// TIA Portal V18 export
// export: Created 2026-06-11T03:43:49.8808703Z, ExportSetting WithDefaults, DisplayName Totally Integrated Automation Portal, DisplayVersion V18, DisplayName TIA Portal Openness, DisplayVersion V18, DisplayName TIA Portal Version Control Interface, DisplayVersion V18, DisplayName STEP 7 Professional, DisplayVersion V18, DisplayName STEP 7 Safety, DisplayVersion V18, DisplayName WinCC Professional, DisplayVersion V18
Screen "03_PID_Muc_Nuoc"  800x600, Number=3
  ScreenLayer 
    GraphicView "Graphic view_1" at 0,0 size 800x600  Picture=Màn PID và nước
    Button "Button_1" at 27,529 size 107x46  Mode=Text, TextOff="TỔNG QUAN", TextOn="Text"
      on Click: ActivateScreen(Screen name := 01_Tong_Quan, Object number := 0)
    Button "Button_2" at 153,529 size 107x46  Mode=Text, TextOff="VẬN HÀNH", TextOn="Text"
      on Click: ActivateScreen(Screen name := 02_Van_Hanh, Object number := 0)
    Button "Button_4" at 409,528 size 107x46  Mode=Text, TextOff="TREND", TextOn="Text"
      on Click: ActivateScreen(Screen name := 04_Trend, Object number := 0)
    Button "Button_5" at 537,528 size 107x46  Mode=Text, TextOff="CẢNH BÁO", TextOn="Text"
      on Click: ActivateScreen(Screen name := 05_Canh_Bao_IO, Object number := 0)
    TextField "Text field_1" at 223,5 size 340x31  Text="MÀN HÌNH 3 - PID MỨC NƯỚC"
    Circle "Circle_3" at 677,3 size 39x39
      RangeAppearanceAnimation "RangeAppearanceAnimation"
        tag bSystemRun
        0..0: back #d9d9d9, fore #181c31
        1..1: back #00ff00, fore #181c31
    Circle "Circle_2" at 718,3 size 39x39
      RangeAppearanceAnimation "RangeAppearanceAnimation"
        tag Loi_He_Thong
        0..0: back #d9d9d9, fore #181c31
        1..1: back #ff0000, fore #181c31
    Circle "Circle_1" at 759,3 size 39x39
      RangeAppearanceAnimation "RangeAppearanceAnimation"
        tag bCheDoMoPhong
        0..0: back #d9d9d9, fore #181c31
        1..1: back #0000ff, fore #181c31
    TextField "Text field_3" at 717,42 size 43x22  Text="Fault"
    TextField "Text field_2" at 679,42 size 34x22  Text="Run"
    TextField "Text field_4" at 760,42 size 33x22  Text="Sim"
    Bar "Bar_1" at 99,165 size 93x220  CountSubDivisions=1, IntegerDigits=2, LargeTickLabelingStep=1, MaximumValue=0.5, Precision=1
      ProcessValue := Muc_Nuoc_PV
    TextField "Text field_6" at 374,80 size 30x22  Text="SP:"
    IOField "I/O field_1" at 407,82 size 37x18  DataFormat=Decimal, FormatPattern=9.9, Mode=InOutput
      ProcessValue := Muc_Nuoc_SP
    TextField "Text field_20" at 445,79 size 18x22  Text="m"
    TextField "Text field_5" at 373,112 size 30x22  Text="PV:"
    IOField "I/O field_2" at 406,114 size 40x19  DataFormat=Decimal, FormatPattern=9.9, Mode=InOutput
      ProcessValue := Muc_Nuoc_PV
    TextField "Text field_7" at 445,111 size 18x22  Text="m"
    TextField "Text field_8" at 373,144 size 32x22  Text="OP:"
    IOField "I/O field_3" at 401,144 size 49x24  DataFormat=Decimal, FormatPattern=99.9, Mode=Output
      ProcessValue := Van_Xa_OP
    TextField "Text field_9" at 443,145 size 23x22  Text="%"
    TextField "Text field_10" at 373,177 size 29x22  Text="Kp:"
    TextField "Text field_11" at 373,209 size 24x22  Text="Ti:"
    TextField "Text field_12" at 373,241 size 28x22  Text="Td:"
    IOField "I/O field_4" at 407,179 size 49x19  DataFormat=Decimal, FormatPattern=999.9, Mode=InOutput
      ProcessValue := PID_Compact_1_sRet_r_Ctrl_Gain
    IOField "I/O field_5" at 396,211 size 61x19  DataFormat=Decimal, FormatPattern=9999.9, Mode=InOutput
      ProcessValue := PID_Compact_1_sRet_r_Ctrl_Ti
    TextField "Text field_13" at 453,209 size 13x22  Text="s"
    IOField "I/O field_6" at 406,243 size 40x19  DataFormat=Decimal, FormatPattern=9.9, Mode=Output
      ProcessValue := PID_Compact_1_sRet_r_Ctrl_Td
    TextField "Text field_14" at 447,239 size 13x22  Text="s"
    Circle "Circle_4" at 486,198 size 25x25
      RangeAppearanceAnimation "RangeAppearanceAnimation"
        tag PID_Level_Enable
        0..0: back #d9d9d9, fore #181c31
        1..1: back #00ff00, fore #000000
    Circle "Circle_5" at 522,199 size 25x25
      RangeAppearanceAnimation "RangeAppearanceAnimation"
        tag Bom_Lam_Mat_M
        0..0: back #d9d9d9, fore #181c31
        1..1: back #00ccff, fore #181c31
    Circle "Circle_6" at 559,199 size 24x24
      RangeAppearanceAnimation "RangeAppearanceAnimation"
        tag Nut_EStop_HMI
        0..0: back #d9d9d9, fore #181c31
        1..1: back #00ff00, fore #181c31
    Button "Button_6" at 489,77 size 93x37  Mode=Text, TextOff="AUTO", TextOn="Text"
      RangeAppearanceAnimation "RangeAppearanceAnimation"
        tag PID_Level_Enable
        0..0: back #636571, fore #ffffff
        1..1: back #00ff00, fore #000000
      on Click: SetBit(Tag := PID_Level_Enable)
    Button "Button_7" at 489,147 size 93x37  Mode=Text, TextOff="MANUAL", TextOn="Text"
      RangeAppearanceAnimation "RangeAppearanceAnimation"
        tag PID_Level_Enable
        0..0: back #ffff00, fore #000000
        1..1: back #969696, fore #ffffff
      on Click: ResetBit(Tag := PID_Level_Enable)
    Rectangle "Rectangle_1" at 484,225 size 32x40
    TextField "Text field_15" at 481,231 size 36x24  Text="PID ENABLE"
    Rectangle "Rectangle_2" at 518,225 size 32x40
    Rectangle "Rectangle_3" at 553,225 size 32x40
    TextField "Text field_16" at 520,231 size 28x24  Text="PUMP OK"
    TextField "Text field_17" at 553,232 size 31x24  Text="ESTOP OK"
    Circle "Circle_7" at 752,169 size 13x13
      RangeAppearanceAnimation "RangeAppearanceAnimation"
        tag PID_Level_Enable
        0..0: back #d9d9d9, fore #181c31
        1..1: back #00ff00, fore #000000, flashing
    Circle "Circle_8" at 603,170 size 13x13
      RangeAppearanceAnimation "RangeAppearanceAnimation"
        tag PID_Level_Enable
        0..0: back #d9d9d9, fore #181c31
        1..1: back #00ff00, fore #000000, flashing
    TextField "Text field_18" at 624,206 size 121x18  Text="Độ mở van thực tế"
    IOField "I/O field_7" at 661,222 size 43x18  DataFormat=Decimal, FormatPattern=99.9, Mode=InOutput
      ProcessValue := Van_Xa_OP
    TextField "Text field_19" at 702,221 size 23x22  Text="%"
    TextField "Text field_21" at 652,248 size 65x18  Text="DAC RAW"
    IOField "I/O field_8" at 662,256 size 49x24  DataFormat=Decimal, FormatPattern=99999, Mode=Output
      ProcessValue := Van_Xa_OP
    Rectangle "Rectangle_8" at 278,526 size 114x52
    Button "Button_3" at 281,529 size 107x46  Mode=Text, TextOff="PID MỨC", TextOn="Text"
      on Click: ActivateScreen(Screen name := , Object number := 0)
    Button "Button_8" at 686,535 size 65x30  Mode=Text, TextOff="EXIT", TextOn="Text"
      on Click: StopRuntime(Mode := 0)
